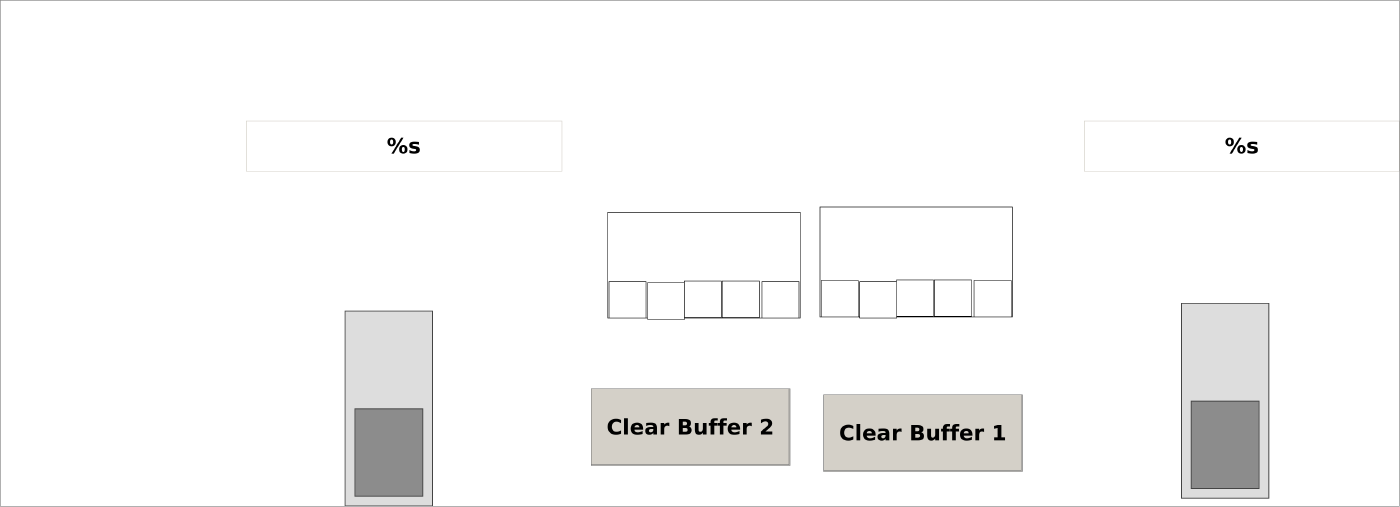
VISUALIZATION Visualization  // 2362x856
    Rectangle (1383,349 325x186)
    Rectangle (1385,473 63x62), invisible if: NOT MAIN.Buffer_1.Places[1]
    Rectangle (1450,475 63x62), invisible if: NOT MAIN.Buffer_1.Places[2]
    Rectangle (1512,472 63x62), invisible if: NOT MAIN.Buffer_1.Places[3]
    Rectangle (1576,472 63x62), invisible if: NOT MAIN.Buffer_1.Places[4]
    Rectangle (1643,473 63x62), invisible if: NOT MAIN.Buffer_1.Places[5]
    Rectangle (1025,358 325x179)
    Rectangle (1027,475 63x62), invisible if: NOT MAIN.Buffer_2.Places[1]
    Rectangle (1092,477 63x62), invisible if: NOT MAIN.Buffer_2.Places[2]
    Rectangle (1154,474 63x62), invisible if: NOT MAIN.Buffer_2.Places[3]
    Rectangle (1218,474 63x62), invisible if: NOT MAIN.Buffer_2.Places[4]
    Rectangle (1285,475 63x62), invisible if: NOT MAIN.Buffer_2.Places[5]
    Button (1389,666 336x130), "Clear Buffer 1"
        OnMouseDown: execute { Main.ClearBuffer_1 := TRUE; }
    Button (997,656 336x130), "Clear Buffer 2"
        OnMouseDown: execute { Main.ClearBuffer_2 := TRUE; }
    Label (1720,208 348x157)
    Label (1761,218 150x115)
    Textfield (1829,204 533x85), "%s", text variable: MAIN.Mover_1.StatusDisp
    Textfield (415,204 533x85), "%s", text variable: MAIN.Mover_2.StatusDisp
    DipSwitch (1902,510 330x333), variable: MAIN.DisableMover_1, behaviour: TOGGLE, style: Switch-DipSwitch-Gray
    DipSwitch (491,523 330x333), variable: MAIN.DisableMover_2, behaviour: TOGGLE, style: Switch-DipSwitch-Gray
END_VISUALIZATION

(* stored: Version 1.1.0.1, ProductVersion 3.1.4024.12
   Visu Visualization: Id {c942bda6-13e7-43b9-8d22-a6d2654a44a3} *)
